(* IEC 61131-3 sources: codesys-build/examples/frame-assembly/src/publication, 2 files *)

(* ---- GVL_Example.st ---- *)
{attribute 'qualified_only'}
VAR_GLOBAL CONSTANT
	Description : STRING := 'Offline example';
END_VAR

(* ---- PRG_Publish.declaration.st ---- *)
PROGRAM PRG_Publish
VAR
	Heartbeat : UDINT;
END_VAR
